// Mitsubishi GX Works2 project: BookEX6_3 TypeConv   PLC: Q13UDV

// global labels: Global
VAR_GLOBAL
  bVar0 AT M5000 : BOOL;
  abArray0 AT M5010 : ARRAY [0..49] OF BOOL;
  sStr0 AT D5000 : STRING[199];
  sStr1 AT D5100 : STRING[199];
  sStr2 AT D5200 : STRING[199];
  sStr3 AT D5300 : STRING[199];
  sStr4 AT D5400 : STRING[199];
  sStr5 AT D5500 : STRING[199];
  sStr6 AT D5600 : STRING[199];
  sStr7 AT D5700 : STRING[199];
  sStr8 AT D5800 : STRING[199];
  sStr9 AT D5900 : STRING[199];
  iVar0 AT D4500 : INT;
  iVar1 AT D4501 : INT;
  iVar2 AT D4502 : INT;
  iVar3 AT D4503 : INT;
  iVar4 AT D4504 : INT;
  iVar5 AT D4505 : INT;
  iVar6 AT D4506 : INT;
  iVar7 AT D4507 : INT;
  iVar8 AT D4508 : INT;
  iVar9 AT D4509 : INT;
  dVar0 AT D4510 : DINT;
  dVar1 AT D4512 : DINT;
  dVar2 AT D4514 : DINT;
  dVar3 AT D4516 : DINT;
  dVar4 AT D4518 : DINT;
  dVar5 AT D4520 : DINT;
  dVar6 AT D4522 : DINT;
  dVar7 AT D4524 : DINT;
  dVar8 AT D4526 : DINT;
  dVar9 AT D4528 : DINT;
  wVar0 AT D4530 : WORD;
  wVar1 AT D4531 : WORD;
  wVar2 AT D4532 : WORD;
  wVar3 AT D4533 : WORD;
  wVar4 AT D4534 : WORD;
  wVar5 AT D4535 : WORD;
  wVar6 AT D4536 : WORD;
  wVar7 AT D4537 : WORD;
  wVar8 AT D4538 : WORD;
  wVar9 AT D4539 : WORD;
  dwVar0 AT D4540 : DWORD;
  dwVar1 AT D4542 : DWORD;
  dwVar2 AT D4544 : DWORD;
  dwVar3 AT D4546 : DWORD;
  dwVar4 AT D4548 : DWORD;
  dwVar5 AT D4550 : DWORD;
  dwVar6 AT D4552 : DWORD;
  dwVar7 AT D4554 : DWORD;
  dwVar8 AT D4556 : DWORD;
  dwVar9 AT D4558 : DWORD;
  fsVar0 AT D4560 : REAL;
  fsVar1 AT D4562 : REAL;
  fsVar2 AT D4564 : REAL;
  fsVar3 AT D4566 : REAL;
  fsVar4 AT D4568 : REAL;
  fsVar5 AT D4570 : REAL;
  fsVar6 AT D4572 : REAL;
  fsVar7 AT D4574 : REAL;
  fsVar8 AT D4576 : REAL;
  fsVar9 AT D4578 : REAL;
  fdVar0 AT D4580 : LREAL;
  tTime0 AT D4620 : TIME;
  tTime1 AT D4622 : TIME;
  tTime2 AT D4624 : TIME;
  tTime3 AT D4626 : TIME;
  tTime4 AT D4628 : TIME;
  tTime5 AT D4630 : TIME;
  tTime6 AT D4632 : TIME;
  tTime7 AT D4634 : TIME;
  tTime8 AT D4636 : TIME;
  tTime9 AT D4638 : TIME;
  tTime10 AT D4640 : TIME;
  bVar1 AT M5001 : BOOL;
  bVar2 AT M5002 : BOOL;
  bVar3 AT M5003 : BOOL;
  bVar4 AT M5004 : BOOL;
  bVar5 AT M5005 : BOOL;
  bVar6 AT M5006 : BOOL;
  bVar7 AT M5007 : BOOL;
  bVar8 AT M5008 : BOOL;
  bVar9 AT M5009 : BOOL;
  abArray1 AT M5060 : ARRAY [0..49] OF BOOL;
  abArray2 AT M5110 : ARRAY [0..49] OF BOOL;
  abArray3 AT M5160 : ARRAY [0..49] OF BOOL;
  abArray4 AT M5210 : ARRAY [0..49] OF BOOL;
  abArray5 AT M5260 : ARRAY [0..49] OF BOOL;
  abArray6 AT M5310 : ARRAY [0..49] OF BOOL;
  abArray7 AT M5360 : ARRAY [0..49] OF BOOL;
  abArray8 AT M5410 : ARRAY [0..49] OF BOOL;
  abArray9 AT M5460 : ARRAY [0..49] OF BOOL;
  fdVar1 AT D4584 : LREAL;
  fdVar2 AT D4588 : LREAL;
  fdVar3 AT D4592 : LREAL;
  fdVar4 AT D4596 : LREAL;
  fdVar5 AT D4600 : LREAL;
  fdVar6 AT D4604 : LREAL;
  fdVar7 AT D4608 : LREAL;
  fdVar8 AT D4612 : LREAL;
  fdVar9 AT D4616 : LREAL;
  adwD10 AT D10 : ARRAY [0..9] OF DWORD;
  awD10 AT D10 : ARRAY [0..19] OF WORD;
  abM10 AT M10 : ARRAY [0..19] OF BOOL;
END_VAR
// user libraries (not included): HMI

FUNCTION Bit2Word
VAR_INPUT
  Bit0 : BOOL;
  Bit1 : BOOL;
  Bit2 : BOOL;
  Bit3 : BOOL;
  Bit4 : BOOL;
  Bit5 : BOOL;
  Bit6 : BOOL;
  Bit7 : BOOL;
END_VAR
;
Bit2Word := SHL(SHL(SHL(SHL(SHL(SHL(SHL(BOOL_TO_WORD(Bit7),1) OR BOOL_TO_WORD(Bit6),1) 
                     OR BOOL_TO_WORD(Bit5),1) OR BOOL_TO_WORD(Bit4),1)
	                 OR BOOL_TO_WORD(Bit3),1) OR BOOL_TO_WORD(Bit2),1) 
	                 OR BOOL_TO_WORD(Bit1),1) OR BOOL_TO_WORD(Bit0);
END_FUNCTION

FUNCTION CopyBitWORD
VAR_INPUT
  ws_IN : WORD;
  is_POS : INT;
  wd_IN : WORD;
  id_POS : INT;
END_VAR
VAR
  b_DATA : BOOL;
  w_DATA : WORD;
END_VAR
;
w_DATA := ws_IN;
SFR(TRUE, is_POS, w_DATA);
b_DATA:= ( w_DATA AND 16#0001) > 0;	
w_DATA := H0001;
SFL(TRUE, id_POS, w_DATA);	
IF b_DATA THEN
	CopyBitWORD := wd_IN OR w_DATA;
ELSE
	CopyBitWORD := wd_IN AND (NOT w_DATA);
END_IF;
END_FUNCTION

FUNCTION GetBitWORD
VAR_INPUT
  w_IN : WORD;
  i_POS : INT;
END_VAR
VAR
  w_DATA : WORD;
END_VAR
;
w_DATA := w_IN;
SFR(TRUE, i_POS, w_DATA);
GetBitWORD := ( w_DATA AND 16#0001) > 0;
END_FUNCTION

FUNCTION SetBitWORD
VAR_INPUT
  w_IN : WORD;
  b_DAT : BOOL;
  i_POS : INT;
END_VAR
VAR
  w_DATA : WORD;
END_VAR
;
w_DATA := H0001;
SFL(TRUE, i_POS, w_DATA);	
IF b_DAT THEN
	SetBitWORD := w_IN OR w_DATA;
ELSE
	SetBitWORD := w_IN AND (NOT w_DATA);
END_IF;
END_FUNCTION

FUNCTION ToggBitWORD
VAR_INPUT
  w_IN : WORD;
  i_POS : INT;
END_VAR
VAR
  w_DATA : WORD;
END_VAR
;
w_DATA := H0001;
SFL(TRUE, i_POS, w_DATA);	
ToggBitWORD := w_IN XOR w_DATA;
END_FUNCTION

FUNCTION_BLOCK Word2Bit
VAR_INPUT
  IN : WORD;
END_VAR
VAR_OUTPUT
  Bit0 : BOOL;
  Bit1 : BOOL;
  Bit2 : BOOL;
  Bit3 : BOOL;
  Bit4 : BOOL;
  Bit5 : BOOL;
  Bit6 : BOOL;
  Bit7 : BOOL;
  Bit8 : BOOL;
  Bit9 : BOOL;
  Bit10 : BOOL;
  Bit11 : BOOL;
  Bit12 : BOOL;
  Bit13 : BOOL;
  Bit14 : BOOL;
  Bit15 : BOOL;
END_VAR
 
Bit0 := WORD_TO_BOOL(IN AND 16#0001);
Bit1 := WORD_TO_BOOL(SHR(IN AND 16#0002 , 1));
Bit2 := WORD_TO_BOOL(SHR(IN AND 16#0004 , 2));
Bit3 := WORD_TO_BOOL(SHR(IN AND 16#0008 , 3));
Bit4 := WORD_TO_BOOL(SHR(IN AND 16#0010 , 4));
Bit5 := WORD_TO_BOOL(SHR(IN AND 16#0020 , 5));
Bit6 := WORD_TO_BOOL(SHR(IN AND 16#0040 , 6));
Bit7 := WORD_TO_BOOL(SHR(IN AND 16#0080 , 7));
Bit8 := WORD_TO_BOOL(SHR(IN AND 16#0100 , 8));
Bit9 := WORD_TO_BOOL(SHR(IN AND 16#0200 , 9));
Bit10 := WORD_TO_BOOL(SHR(IN AND 16#0400 , 10));
Bit11 := WORD_TO_BOOL(SHR(IN AND 16#0800 , 11));
Bit12 := WORD_TO_BOOL(SHR(IN AND 16#1000 , 12));
Bit13 := WORD_TO_BOOL(SHR(IN AND 16#2000 , 13));
Bit14 := WORD_TO_BOOL(SHR(IN AND 16#4000 , 14));
Bit15 := WORD_TO_BOOL(SHR(IN AND 16#8000 , 15));
END_FUNCTION_BLOCK

PROGRAM ExBIT_INT
(* structured ladder/FBD written out as ST: instructions are called as NAME(EN, inputs, outputs); _pN, _eN, _tN stand for wires *)
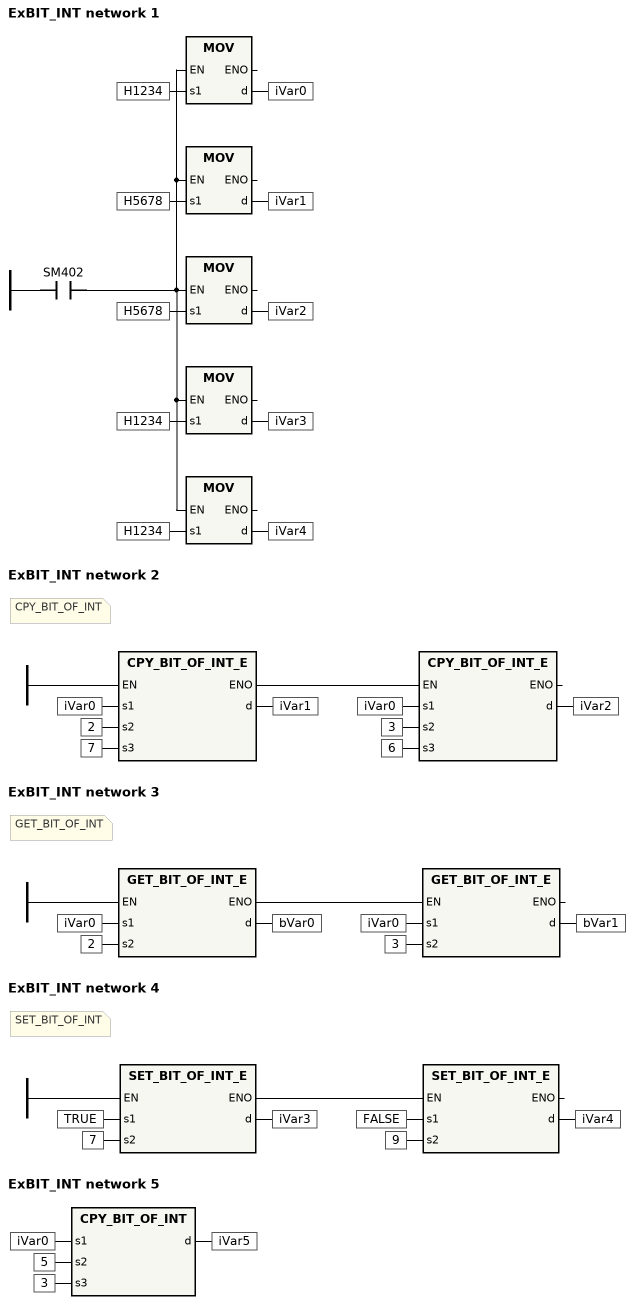
(* network 1 *)
MOV(SM402, H1234, iVar0);
MOV(SM402, H5678, iVar1);
MOV(SM402, H5678, iVar2);
MOV(SM402, H1234, iVar3);
MOV(SM402, H1234, iVar4);
(* network 2 *)
(* CPY_BIT_OF_INT *)
_e1 := CPY_BIT_OF_INT_E(TRUE, iVar0, 2, 7, iVar1);
CPY_BIT_OF_INT_E(_e1, iVar0, 3, 6, iVar2);
(* network 3 *)
(* GET_BIT_OF_INT *)
_e1 := GET_BIT_OF_INT_E(TRUE, iVar0, 2, bVar0);
GET_BIT_OF_INT_E(_e1, iVar0, 3, bVar1);
(* network 4 *)
(* SET_BIT_OF_INT *)
_e1 := SET_BIT_OF_INT_E(TRUE, TRUE, 7, iVar3);
SET_BIT_OF_INT_E(_e1, FALSE, 9, iVar4);
(* network 5 *)
iVar5 := CPY_BIT_OF_INT(iVar0, 5, 3);
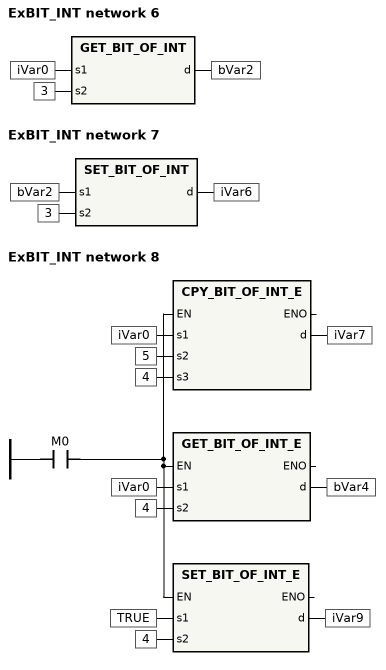
(* network 6 *)
bVar2 := GET_BIT_OF_INT(iVar0, 3);
(* network 7 *)
iVar6 := SET_BIT_OF_INT(bVar2, 3);
(* network 8 *)
CPY_BIT_OF_INT_E(M0, iVar0, 5, 4, iVar7);
GET_BIT_OF_INT_E(M0, iVar0, 4, bVar4);
SET_BIT_OF_INT_E(M0, TRUE, 4, iVar9);
END_PROGRAM

PROGRAM ExBIT_WORD
(* structured ladder/FBD written out as ST: instructions are called as NAME(EN, inputs, outputs); _pN, _eN, _tN stand for wires *)
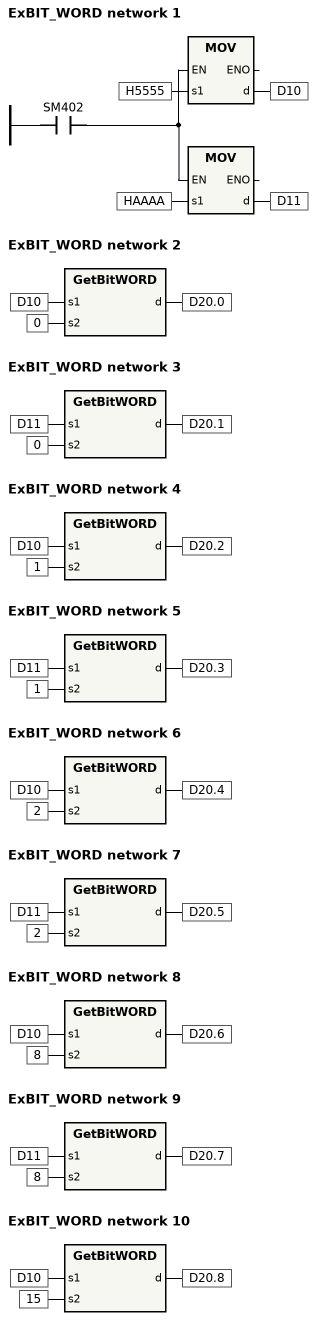
(* network 1 *)
MOV(SM402, H5555, D10);
MOV(SM402, HAAAA, D11);
(* network 2 *)
D20.0 := GetBitWORD(D10, 0);
(* network 3 *)
D20.1 := GetBitWORD(D11, 0);
(* network 4 *)
D20.2 := GetBitWORD(D10, 1);
(* network 5 *)
D20.3 := GetBitWORD(D11, 1);
(* network 6 *)
D20.4 := GetBitWORD(D10, 2);
(* network 7 *)
D20.5 := GetBitWORD(D11, 2);
(* network 8 *)
D20.6 := GetBitWORD(D10, 8);
(* network 9 *)
D20.7 := GetBitWORD(D11, 8);
(* network 10 *)
D20.8 := GetBitWORD(D10, 15);
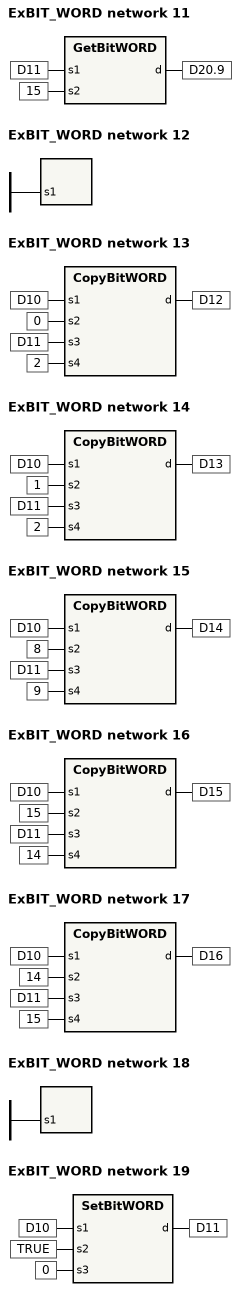
(* network 11 *)
D20.9 := GetBitWORD(D11, 15);
(* network 12 *)
(* element kind 10  <- TRUE *)
(* network 13 *)
D12 := CopyBitWORD(D10, 0, D11, 2);
(* network 14 *)
D13 := CopyBitWORD(D10, 1, D11, 2);
(* network 15 *)
D14 := CopyBitWORD(D10, 8, D11, 9);
(* network 16 *)
D15 := CopyBitWORD(D10, 15, D11, 14);
(* network 17 *)
D16 := CopyBitWORD(D10, 14, D11, 15);
(* network 18 *)
(* element kind 10  <- TRUE *)
(* network 19 *)
D11 := SetBitWORD(D10, TRUE, 0);
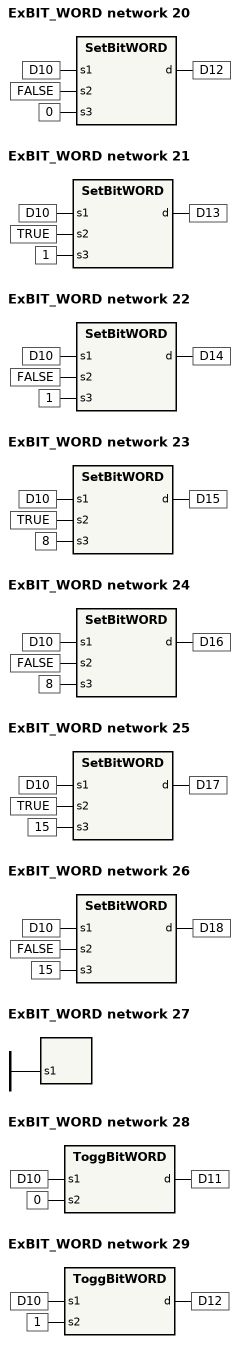
(* network 20 *)
D12 := SetBitWORD(D10, FALSE, 0);
(* network 21 *)
D13 := SetBitWORD(D10, TRUE, 1);
(* network 22 *)
D14 := SetBitWORD(D10, FALSE, 1);
(* network 23 *)
D15 := SetBitWORD(D10, TRUE, 8);
(* network 24 *)
D16 := SetBitWORD(D10, FALSE, 8);
(* network 25 *)
D17 := SetBitWORD(D10, TRUE, 15);
(* network 26 *)
D18 := SetBitWORD(D10, FALSE, 15);
(* network 27 *)
(* element kind 10  <- TRUE *)
(* network 28 *)
D11 := ToggBitWORD(D10, 0);
(* network 29 *)
D12 := ToggBitWORD(D10, 1);
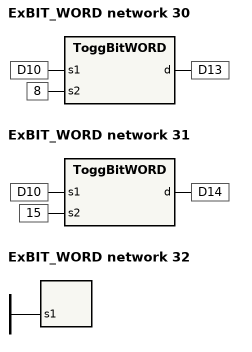
(* network 30 *)
D13 := ToggBitWORD(D10, 8);
(* network 31 *)
D14 := ToggBitWORD(D10, 15);
(* network 32 *)
(* element kind 10  <- TRUE *)
END_PROGRAM

PROGRAM ExBITARR
VAR
  Word2Bit_1 : Word2Bit;
END_VAR
VAR CONSTANT
  num1 : INT := 4;
  num2 : INT := 1;
END_VAR
VAR
  INT2Bit_1 : INT2Bit;
  Flag0 : BOOL;
  Flag1 : BOOL;
  Flag2 : BOOL;
  Flag3 : BOOL;
  Flag4 : BOOL;
  Flag5 : BOOL;
  Flag6 : BOOL;
  Flag7 : BOOL;
  Flag8 : BOOL;
  Flag9 : BOOL;
  Flag10 : BOOL;
  Flag11 : BOOL;
  Flag12 : BOOL;
  Flag13 : BOOL;
  Flag14 : BOOL;
  Flag15 : BOOL;
  abTemp : ARRAY [0..49] OF BOOL;
END_VAR
(* structured ladder/FBD written out as ST: instructions are called as NAME(EN, inputs, outputs); _pN, _eN, _tN stand for wires *)
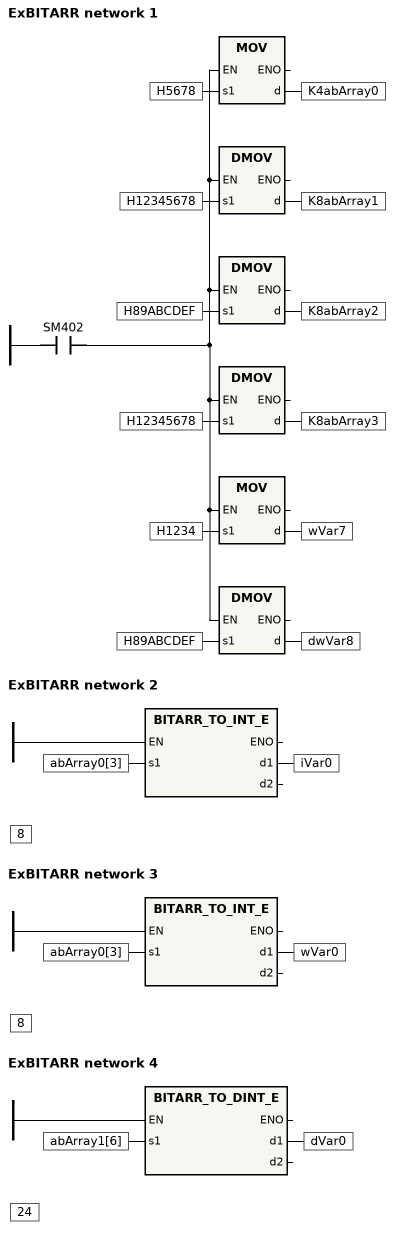
(* network 1 *)
MOV(SM402, H5678, K4abArray0);
DMOV(SM402, H12345678, K8abArray1);
DMOV(SM402, H89ABCDEF, K8abArray2);
DMOV(SM402, H12345678, K8abArray3);
MOV(SM402, H1234, wVar7);
DMOV(SM402, H89ABCDEF, dwVar8);
(* network 2 *)
BITARR_TO_INT_E(TRUE, abArray0[3], iVar0, _open);
(* not connected to any output: 8 *)
(* network 3 *)
BITARR_TO_INT_E(TRUE, abArray0[3], wVar0, _open);
(* not connected to any output: 8 *)
(* network 4 *)
BITARR_TO_DINT_E(TRUE, abArray1[6], dVar0, _open);
(* not connected to any output: 24 *)
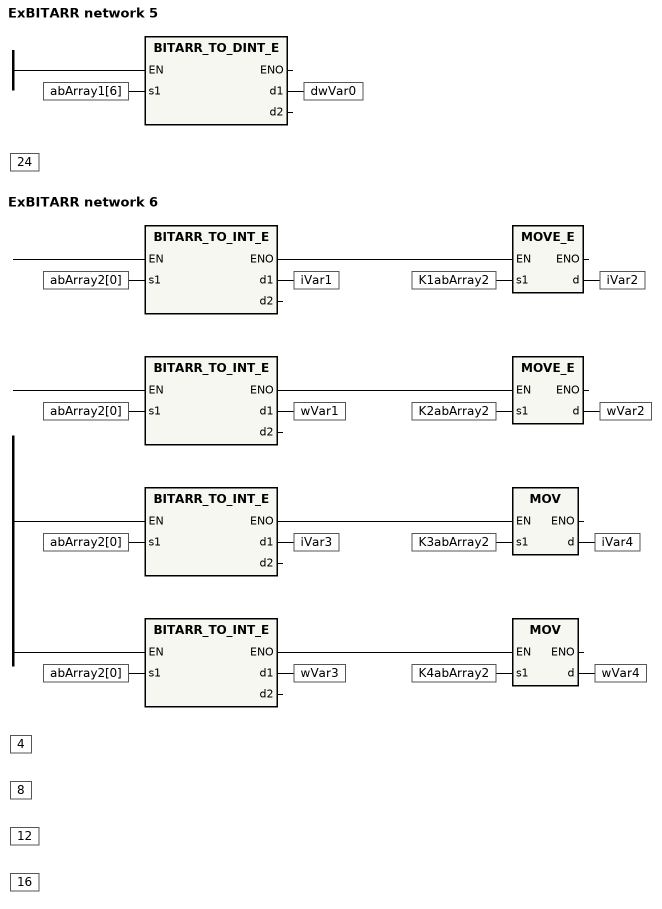
(* network 5 *)
BITARR_TO_DINT_E(TRUE, abArray1[6], dwVar0, _open);
(* not connected to any output: 24 *)
(* network 6 *)
_e1 := BITARR_TO_INT_E(TRUE, abArray2[0], iVar1, _open);
MOVE_E(_e1, K1abArray2, iVar2);
_e2 := BITARR_TO_INT_E(TRUE, abArray2[0], wVar1, _open);
MOVE_E(_e2, K2abArray2, wVar2);
_e3 := BITARR_TO_INT_E(TRUE, abArray2[0], iVar3, _open);
MOV(_e3, K3abArray2, iVar4);
_e4 := BITARR_TO_INT_E(TRUE, abArray2[0], wVar3, _open);
MOV(_e4, K4abArray2, wVar4);
(* not connected to any output: 4, 8, 12, 16 *)
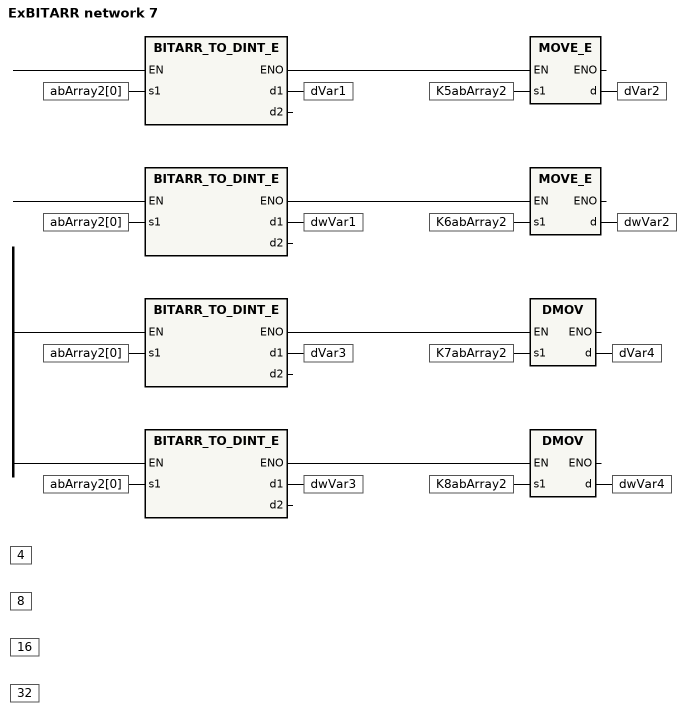
(* network 7 *)
_e1 := BITARR_TO_DINT_E(TRUE, abArray2[0], dVar1, _open);
MOVE_E(_e1, K5abArray2, dVar2);
_e2 := BITARR_TO_DINT_E(TRUE, abArray2[0], dwVar1, _open);
MOVE_E(_e2, K6abArray2, dwVar2);
_e3 := BITARR_TO_DINT_E(TRUE, abArray2[0], dVar3, _open);
DMOV(_e3, K7abArray2, dVar4);
_e4 := BITARR_TO_DINT_E(TRUE, abArray2[0], dwVar3, _open);
DMOV(_e4, K8abArray2, dwVar4);
(* not connected to any output: 4, 8, 16, 32 *)
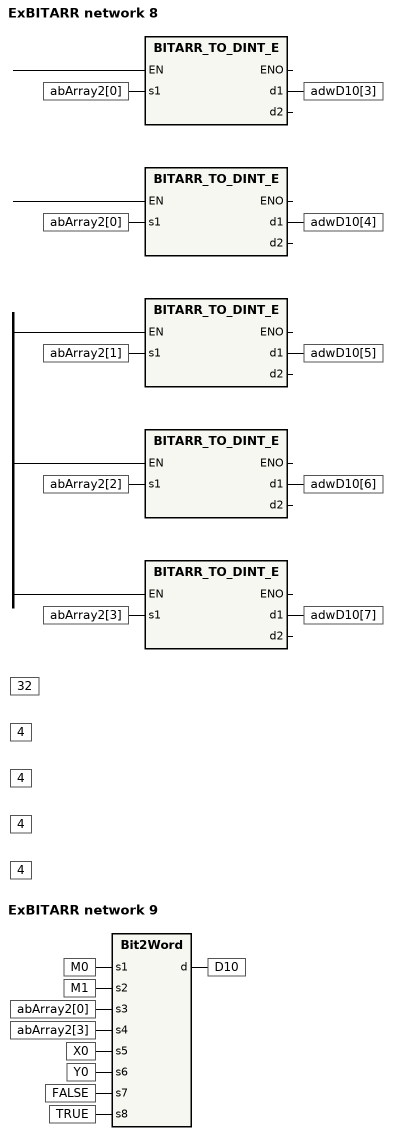
(* network 8 *)
BITARR_TO_DINT_E(TRUE, abArray2[0], adwD10[3], _open);
BITARR_TO_DINT_E(TRUE, abArray2[0], adwD10[4], _open);
BITARR_TO_DINT_E(TRUE, abArray2[1], adwD10[5], _open);
BITARR_TO_DINT_E(TRUE, abArray2[2], adwD10[6], _open);
BITARR_TO_DINT_E(TRUE, abArray2[3], adwD10[7], _open);
(* not connected to any output: 32, 4, 4, 4, 4 *)
(* network 9 *)
D10 := Bit2Word(M0, M1, abArray2[0], abArray2[3], X0, Y0, FALSE, TRUE);
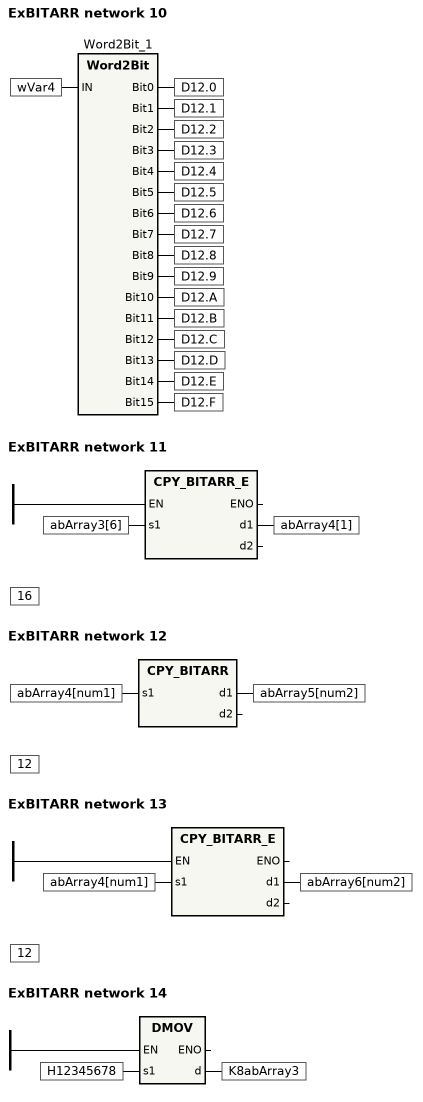
(* network 10 *)
Word2Bit_1(IN := wVar4, Bit0 => D12.0, Bit1 => D12.1, Bit2 => D12.2, Bit3 => D12.3, Bit4 => D12.4, Bit5 => D12.5, Bit6 => D12.6, Bit7 => D12.7, Bit8 => D12.8, Bit9 => D12.9, Bit10 => D12.A, Bit11 => D12.B, Bit12 => D12.C, Bit13 => D12.D, Bit14 => D12.E, Bit15 => D12.F);
(* network 11 *)
CPY_BITARR_E(TRUE, abArray3[6], abArray4[1], _open);
(* not connected to any output: 16 *)
(* network 12 *)
abArray5[num2] := CPY_BITARR(abArray4[num1]);
(* not connected to any output: 12 *)
(* network 13 *)
CPY_BITARR_E(TRUE, abArray4[num1], abArray6[num2], _open);
(* not connected to any output: 12 *)
(* network 14 Jmp1: *)
DMOV(TRUE, H12345678, K8abArray3);
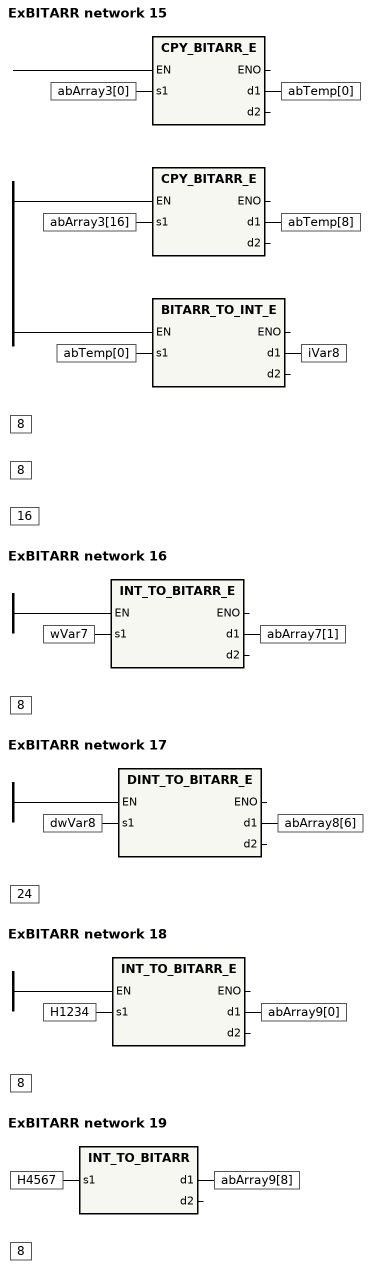
(* network 15 *)
CPY_BITARR_E(TRUE, abArray3[0], abTemp[0], _open);
CPY_BITARR_E(TRUE, abArray3[16], abTemp[8], _open);
BITARR_TO_INT_E(TRUE, abTemp[0], iVar8, _open);
(* not connected to any output: 8, 8, 16 *)
(* network 16 *)
INT_TO_BITARR_E(TRUE, wVar7, abArray7[1], _open);
(* not connected to any output: 8 *)
(* network 17 *)
DINT_TO_BITARR_E(TRUE, dwVar8, abArray8[6], _open);
(* not connected to any output: 24 *)
(* network 18 *)
INT_TO_BITARR_E(TRUE, H1234, abArray9[0], _open);
(* not connected to any output: 8 *)
(* network 19 *)
abArray9[8] := INT_TO_BITARR(H4567);
(* not connected to any output: 8 *)
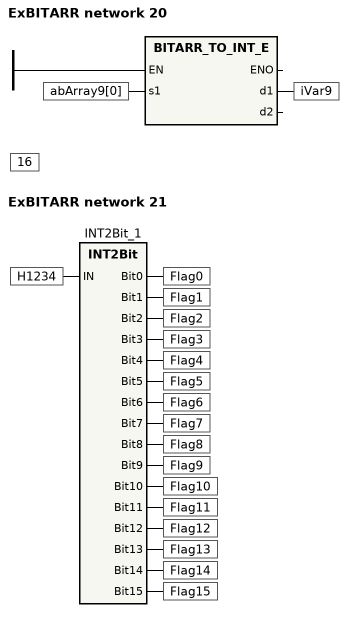
(* network 20 *)
BITARR_TO_INT_E(TRUE, abArray9[0], iVar9, _open);
(* not connected to any output: 16 *)
(* network 21 *)
INT2Bit_1(IN := H1234, Bit0 => Flag0, Bit1 => Flag1, Bit2 => Flag2, Bit3 => Flag3, Bit4 => Flag4, Bit5 => Flag5, Bit6 => Flag6, Bit7 => Flag7, Bit8 => Flag8, Bit9 => Flag9, Bit10 => Flag10, Bit11 => Flag11, Bit12 => Flag12, Bit13 => Flag13, Bit14 => Flag14, Bit15 => Flag15);
END_PROGRAM

PROGRAM ExBOOL_TO
VAR
  GetInt : INT;
  NthBit : INT;
  SetInt : INT;
  SetInt2 : INT;
END_VAR
(* structured ladder/FBD written out as ST: instructions are called as NAME(EN, inputs, outputs); _pN, _eN, _tN stand for wires *)
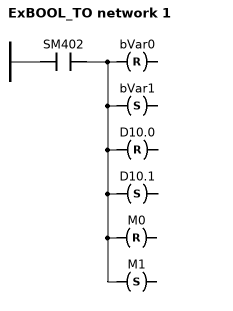
(* network 1 *)
RST(SM402, bVar0);
SET(SM402, bVar1);
RST(SM402, D10.0);
SET(SM402, D10.1);
RST(SM402, M0);
SET(SM402, M1);
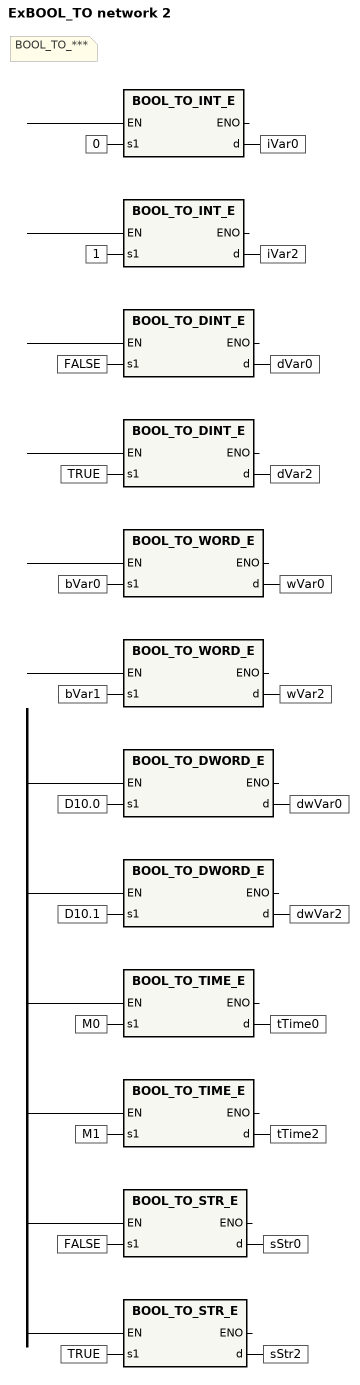
(* network 2 *)
(* BOOL_TO_*** *)
BOOL_TO_INT_E(TRUE, 0, iVar0);
BOOL_TO_INT_E(TRUE, 1, iVar2);
BOOL_TO_DINT_E(TRUE, FALSE, dVar0);
BOOL_TO_DINT_E(TRUE, TRUE, dVar2);
BOOL_TO_WORD_E(TRUE, bVar0, wVar0);
BOOL_TO_WORD_E(TRUE, bVar1, wVar2);
BOOL_TO_DWORD_E(TRUE, D10.0, dwVar0);
BOOL_TO_DWORD_E(TRUE, D10.1, dwVar2);
BOOL_TO_TIME_E(TRUE, M0, tTime0);
BOOL_TO_TIME_E(TRUE, M1, tTime2);
BOOL_TO_STR_E(TRUE, FALSE, sStr0);
BOOL_TO_STR_E(TRUE, TRUE, sStr2);
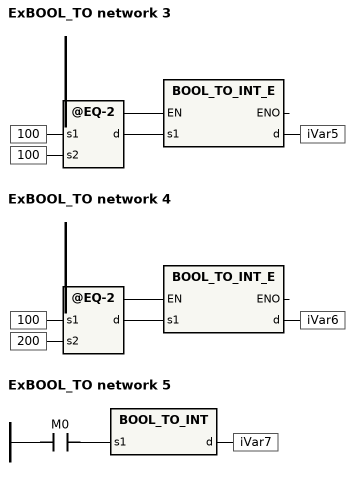
(* network 3 *)
BOOL_TO_INT_E(TRUE, @EQ-2(100, 100), iVar5);
(* network 4 *)
BOOL_TO_INT_E(TRUE, @EQ-2(100, 200), iVar6);
(* network 5 *)
iVar7 := BOOL_TO_INT(M0);
END_PROGRAM

PROGRAM ExBOOL_TO(ST)
(* BOOL_TO_*** *)
bVar0 := FALSE;		M0 := FALSE;  bVar1 := TRUE;		M1 := TRUE;     D10 := 2;
bVar3 := BOOL_TO_INT_E(TRUE, 0, iVar0);							iVar2 := BOOL_TO_INT(1);
bVar3 := BOOL_TO_DINT_E(TRUE, FALSE, dVar0);			dVar2 := BOOL_TO_DINT(TRUE);
bVar3 := BOOL_TO_WORD_E(TRUE, bVar0, wVar0);		wVar2 := BOOL_TO_WORD(bVar1);
bVar3 := BOOL_TO_DWORD_E(TRUE, D10.0, dwVar0);	dwVar2 := BOOL_TO_DWORD(D10.1);
bVar3 := BOOL_TO_TIME_E(TRUE, M0, tTime0);				tTime2 := BOOL_TO_TIME(M1);
bVar3 := BOOL_TO_STR_E(TRUE, FALSE, sStr0);				sStr2 := BOOL_TO_STR(TRUE);
END_PROGRAM

PROGRAM ExDINT_TO
VAR
  GetInt : INT;
  NthBit : INT;
  SetInt : INT;
  SetInt2 : INT;
END_VAR
(* structured ladder/FBD written out as ST: instructions are called as NAME(EN, inputs, outputs); _pN, _eN, _tN stand for wires *)
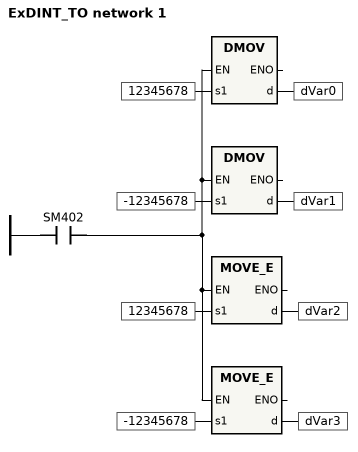
(* network 1 *)
DMOV(SM402, 12345678, dVar0);
DMOV(SM402, -12345678, dVar1);
MOVE_E(SM402, 12345678, dVar2);
MOVE_E(SM402, -12345678, dVar3);
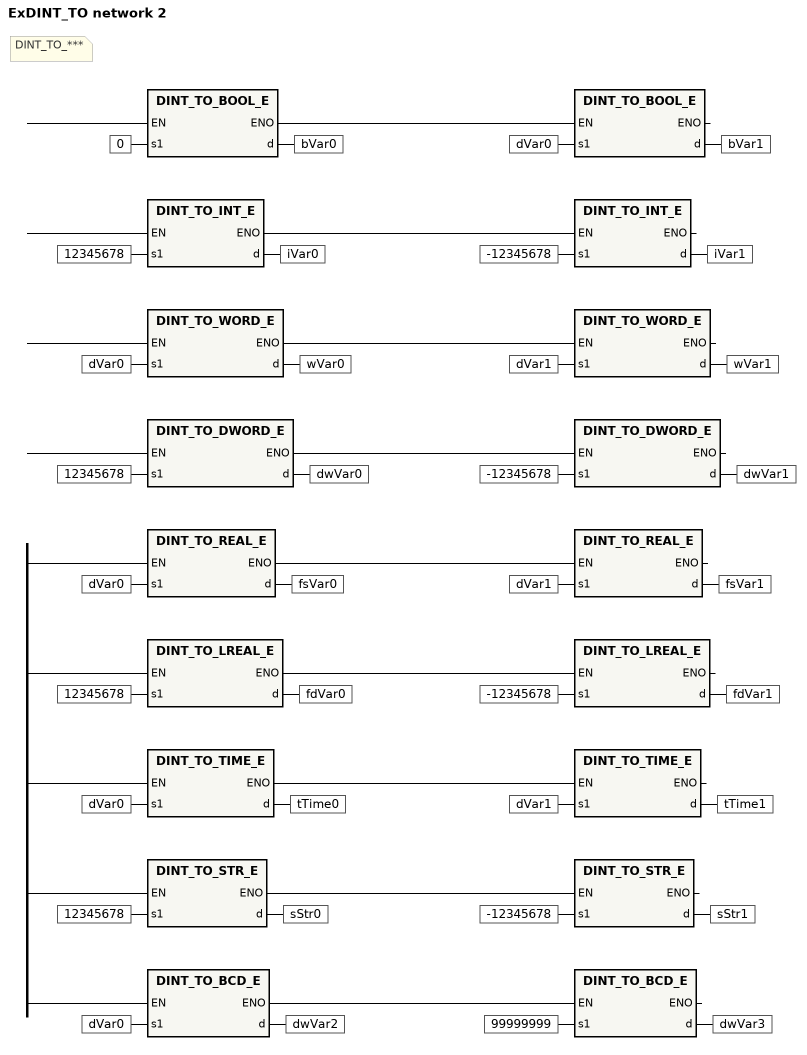
(* network 2 *)
(* DINT_TO_*** *)
_e1 := DINT_TO_BOOL_E(TRUE, 0, bVar0);
DINT_TO_BOOL_E(_e1, dVar0, bVar1);
_e2 := DINT_TO_INT_E(TRUE, 12345678, iVar0);
DINT_TO_INT_E(_e2, -12345678, iVar1);
_e3 := DINT_TO_WORD_E(TRUE, dVar0, wVar0);
DINT_TO_WORD_E(_e3, dVar1, wVar1);
_e4 := DINT_TO_DWORD_E(TRUE, 12345678, dwVar0);
DINT_TO_DWORD_E(_e4, -12345678, dwVar1);
_e5 := DINT_TO_REAL_E(TRUE, dVar0, fsVar0);
DINT_TO_REAL_E(_e5, dVar1, fsVar1);
_e6 := DINT_TO_LREAL_E(TRUE, 12345678, fdVar0);
DINT_TO_LREAL_E(_e6, -12345678, fdVar1);
_e7 := DINT_TO_TIME_E(TRUE, dVar0, tTime0);
DINT_TO_TIME_E(_e7, dVar1, tTime1);
_e8 := DINT_TO_STR_E(TRUE, 12345678, sStr0);
DINT_TO_STR_E(_e8, -12345678, sStr1);
_e9 := DINT_TO_BCD_E(TRUE, dVar0, dwVar2);
DINT_TO_BCD_E(_e9, 99999999, dwVar3);
END_PROGRAM

PROGRAM ExDWORD_TO
VAR
  GetInt : INT;
  NthBit : INT;
  SetInt : INT;
  SetInt2 : INT;
END_VAR
(* structured ladder/FBD written out as ST: instructions are called as NAME(EN, inputs, outputs); _pN, _eN, _tN stand for wires *)
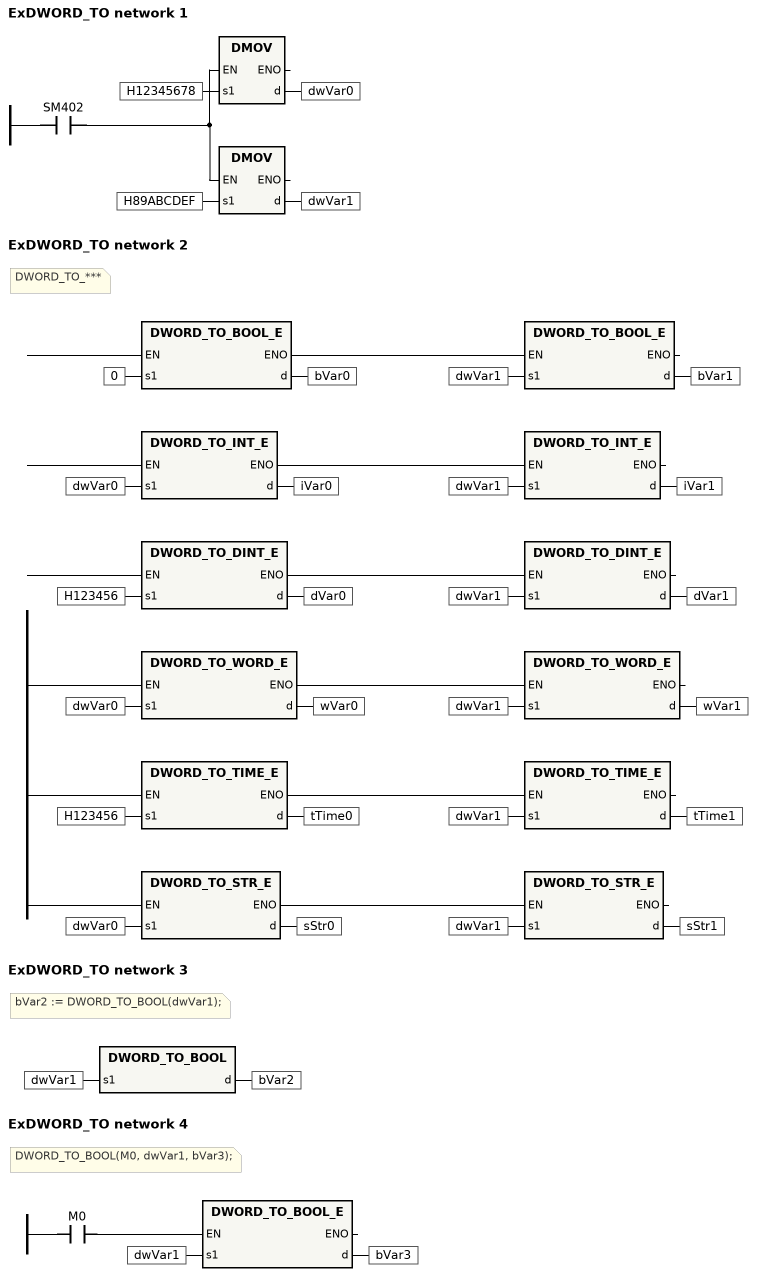
(* network 1 *)
DMOV(SM402, H12345678, dwVar0);
DMOV(SM402, H89ABCDEF, dwVar1);
(* network 2 *)
(* DWORD_TO_*** *)
_e1 := DWORD_TO_BOOL_E(TRUE, 0, bVar0);
DWORD_TO_BOOL_E(_e1, dwVar1, bVar1);
_e2 := DWORD_TO_INT_E(TRUE, dwVar0, iVar0);
DWORD_TO_INT_E(_e2, dwVar1, iVar1);
_e3 := DWORD_TO_DINT_E(TRUE, H123456, dVar0);
DWORD_TO_DINT_E(_e3, dwVar1, dVar1);
_e4 := DWORD_TO_WORD_E(TRUE, dwVar0, wVar0);
DWORD_TO_WORD_E(_e4, dwVar1, wVar1);
_e5 := DWORD_TO_TIME_E(TRUE, H123456, tTime0);
DWORD_TO_TIME_E(_e5, dwVar1, tTime1);
_e6 := DWORD_TO_STR_E(TRUE, dwVar0, sStr0);
DWORD_TO_STR_E(_e6, dwVar1, sStr1);
(* network 3 *)
(* bVar2 := DWORD_TO_BOOL(dwVar1); *)
bVar2 := DWORD_TO_BOOL(dwVar1);
(* network 4 *)
(* DWORD_TO_BOOL(M0, dwVar1, bVar3); *)
DWORD_TO_BOOL_E(M0, dwVar1, bVar3);
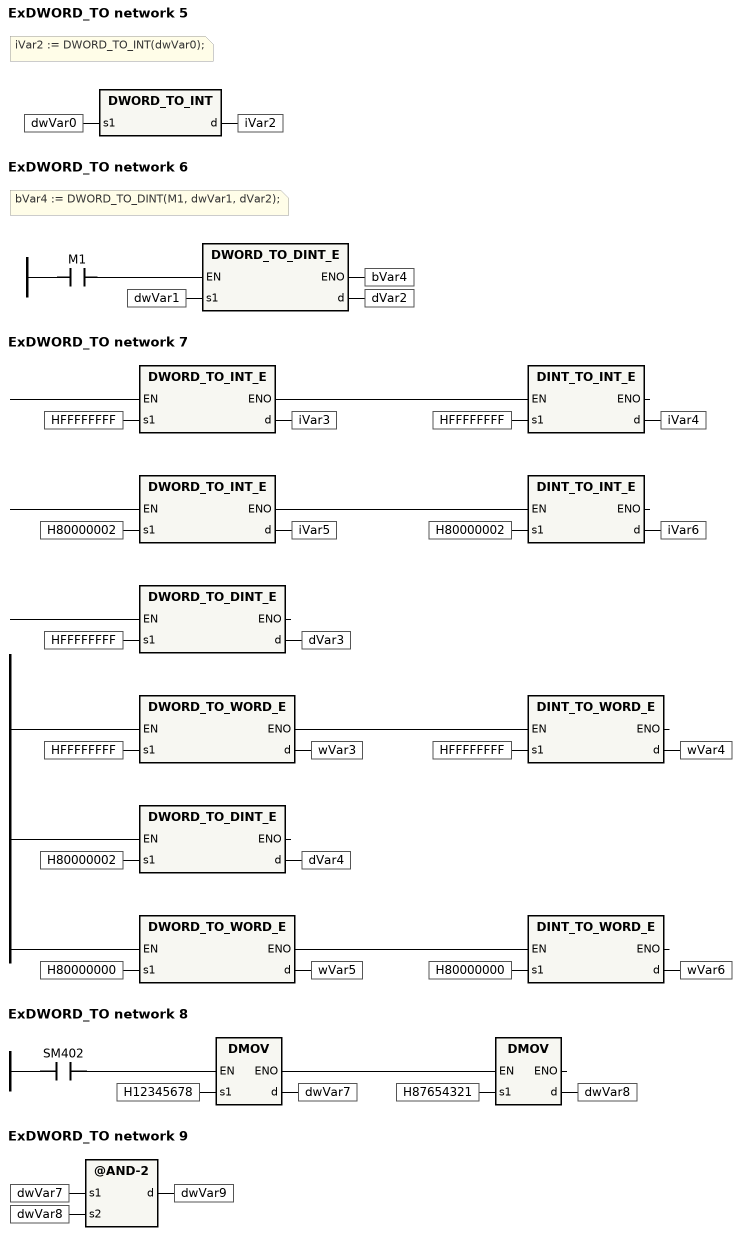
(* network 5 *)
(* iVar2 := DWORD_TO_INT(dwVar0); *)
iVar2 := DWORD_TO_INT(dwVar0);
(* network 6 *)
(* bVar4 := DWORD_TO_DINT(M1, dwVar1, dVar2); *)
_e1 := DWORD_TO_DINT_E(M1, dwVar1, dVar2);
bVar4 := _e1;
(* network 7 *)
_e1 := DWORD_TO_INT_E(TRUE, HFFFFFFFF, iVar3);
DINT_TO_INT_E(_e1, HFFFFFFFF, iVar4);
_e2 := DWORD_TO_INT_E(TRUE, H80000002, iVar5);
DINT_TO_INT_E(_e2, H80000002, iVar6);
DWORD_TO_DINT_E(TRUE, HFFFFFFFF, dVar3);
DWORD_TO_DINT_E(TRUE, H80000002, dVar4);
_e3 := DWORD_TO_WORD_E(TRUE, HFFFFFFFF, wVar3);
DINT_TO_WORD_E(_e3, HFFFFFFFF, wVar4);
_e4 := DWORD_TO_WORD_E(TRUE, H80000000, wVar5);
DINT_TO_WORD_E(_e4, H80000000, wVar6);
(* network 8 *)
_e1 := DMOV(SM402, H12345678, dwVar7);
DMOV(_e1, H87654321, dwVar8);
(* network 9 *)
dwVar9 := @AND-2(dwVar7, dwVar8);
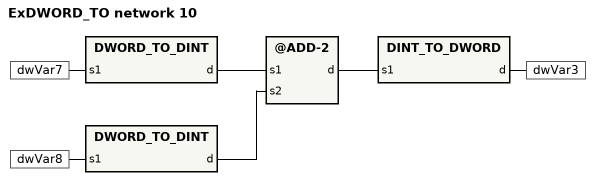
(* network 10 *)
dwVar3 := DINT_TO_DWORD(@ADD-2(DWORD_TO_DINT(dwVar7), DWORD_TO_DINT(dwVar8)));
END_PROGRAM

PROGRAM ExGet_ADDR
(* structured ladder/FBD written out as ST: instructions are called as NAME(EN, inputs, outputs); _pN, _eN, _tN stand for wires *)
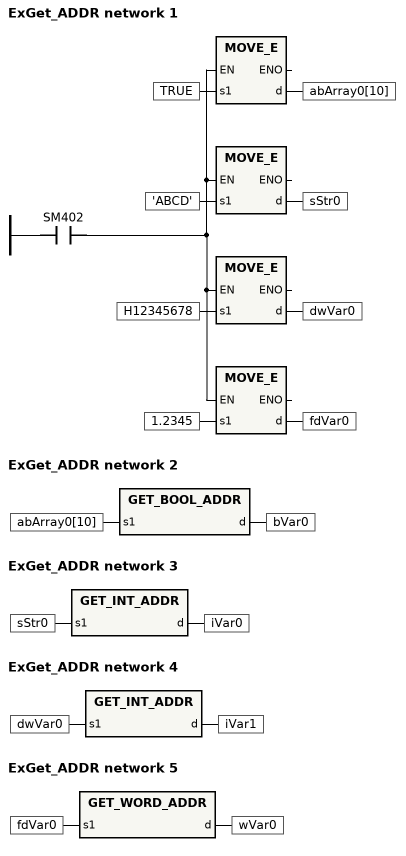
(* network 1 *)
MOVE_E(SM402, TRUE, abArray0[10]);
MOVE_E(SM402, 'ABCD', sStr0);
MOVE_E(SM402, H12345678, dwVar0);
MOVE_E(SM402, 1.2345, fdVar0);
(* network 2 *)
bVar0 := GET_BOOL_ADDR(abArray0[10]);
(* network 3 *)
iVar0 := GET_INT_ADDR(sStr0);
(* network 4 *)
iVar1 := GET_INT_ADDR(dwVar0);
(* network 5 *)
wVar0 := GET_WORD_ADDR(fdVar0);
END_PROGRAM

PROGRAM ExINT_TO
VAR
  GetInt : INT;
  NthBit : INT;
  SetInt : INT;
  SetInt2 : INT;
END_VAR
(* structured ladder/FBD written out as ST: instructions are called as NAME(EN, inputs, outputs); _pN, _eN, _tN stand for wires *)
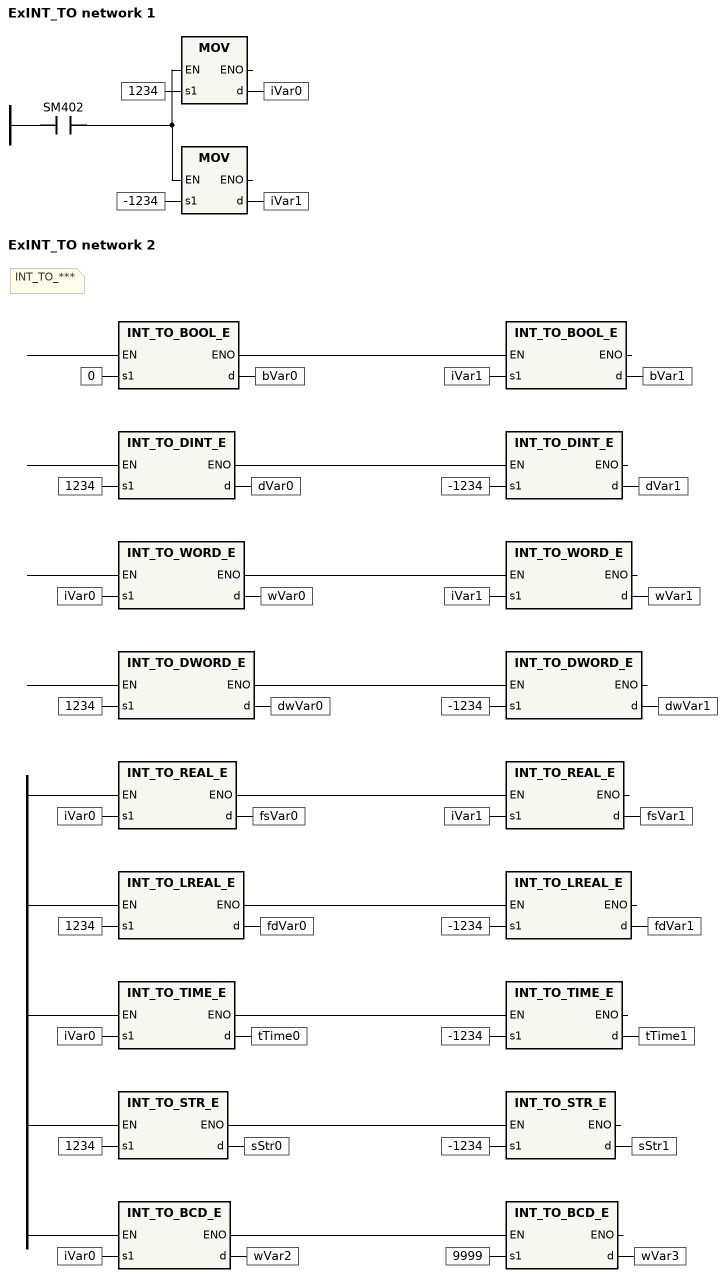
(* network 1 *)
MOV(SM402, 1234, iVar0);
MOV(SM402, -1234, iVar1);
(* network 2 *)
(* INT_TO_*** *)
_e1 := INT_TO_BOOL_E(TRUE, 0, bVar0);
INT_TO_BOOL_E(_e1, iVar1, bVar1);
_e2 := INT_TO_DINT_E(TRUE, 1234, dVar0);
INT_TO_DINT_E(_e2, -1234, dVar1);
_e3 := INT_TO_WORD_E(TRUE, iVar0, wVar0);
INT_TO_WORD_E(_e3, iVar1, wVar1);
_e4 := INT_TO_DWORD_E(TRUE, 1234, dwVar0);
INT_TO_DWORD_E(_e4, -1234, dwVar1);
_e5 := INT_TO_REAL_E(TRUE, iVar0, fsVar0);
INT_TO_REAL_E(_e5, iVar1, fsVar1);
_e6 := INT_TO_LREAL_E(TRUE, 1234, fdVar0);
INT_TO_LREAL_E(_e6, -1234, fdVar1);
_e7 := INT_TO_TIME_E(TRUE, iVar0, tTime0);
INT_TO_TIME_E(_e7, -1234, tTime1);
_e8 := INT_TO_STR_E(TRUE, 1234, sStr0);
INT_TO_STR_E(_e8, -1234, sStr1);
_e9 := INT_TO_BCD_E(TRUE, iVar0, wVar2);
INT_TO_BCD_E(_e9, 9999, wVar3);
END_PROGRAM

PROGRAM ExLREAL_TO
VAR
  GetInt : INT;
  NthBit : INT;
  SetInt : INT;
  SetInt2 : INT;
END_VAR
(* structured ladder/FBD written out as ST: instructions are called as NAME(EN, inputs, outputs); _pN, _eN, _tN stand for wires *)
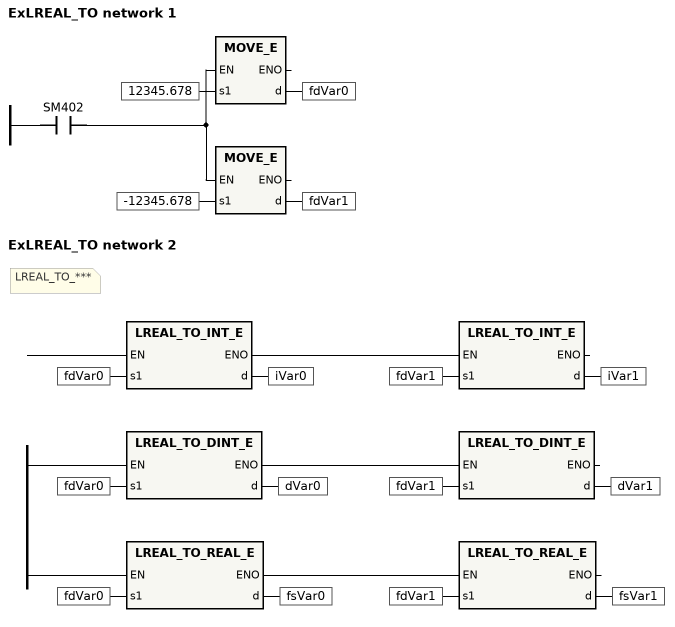
(* network 1 *)
MOVE_E(SM402, 12345.678, fdVar0);
MOVE_E(SM402, -12345.678, fdVar1);
(* network 2 *)
(* LREAL_TO_*** *)
_e1 := LREAL_TO_INT_E(TRUE, fdVar0, iVar0);
LREAL_TO_INT_E(_e1, fdVar1, iVar1);
_e2 := LREAL_TO_DINT_E(TRUE, fdVar0, dVar0);
LREAL_TO_DINT_E(_e2, fdVar1, dVar1);
_e3 := LREAL_TO_REAL_E(TRUE, fdVar0, fsVar0);
LREAL_TO_REAL_E(_e3, fdVar1, fsVar1);
END_PROGRAM

PROGRAM ExREAL_TO
VAR
  GetInt : INT;
  NthBit : INT;
  SetInt : INT;
  SetInt2 : INT;
END_VAR
(* structured ladder/FBD written out as ST: instructions are called as NAME(EN, inputs, outputs); _pN, _eN, _tN stand for wires *)
